// ---- POUs/20_AUTO/ST180/VISU_ST180.TcVIS
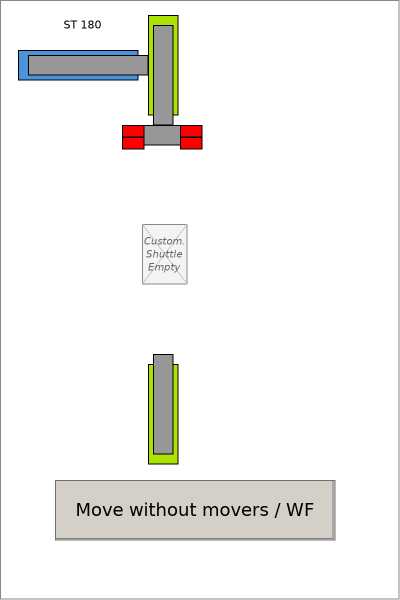
VISUALIZATION VISU_ST180  // 400x600
    Image (142,224 45x60), invisible if: NOT __ISVALIDREF(GVL.st180_aut._Mover), image: Custom.Shuttle Empty
    Rectangle (18,50 120x30)
    Rectangle (28,55 120x20)
        p3560616238: GVL.st180_aut.fb_Pnp.fb_simu_axis180_01Y.rOUT_PixActual
    Rectangle (148,15 30x100)
        p3560616238: GVL.st180_aut.fb_Pnp.fb_simu_axis180_01Y.rOUT_PixActual
    Rectangle (153,25 20x100)
        p2738717112: GVL.st180_aut.fb_Pnp.fb_simu_axis180_02Z.rOUT_PixActual
        p3560616238: GVL.st180_aut.fb_Pnp.fb_simu_axis180_01Y.rOUT_PixActual
    Label (40,15 85x20), "ST 180"
    Rectangle (122,125 80x20)
        p2738717112: GVL.st180_aut.fb_Pnp.fb_simu_axis180_02Z.rOUT_PixActual
        p3560616238: GVL.st180_aut.fb_Pnp.fb_simu_axis180_01Y.rOUT_PixActual
    Ellipse (123,125 20x20), colour toggle: GVL.st180_aut.fb_Pnp.fb_griperLeft.xIN_GS
        p3560616238: GVL.st180_aut.fb_Pnp.fb_simu_axis180_01Y.rOUT_PixActual
        p2738717112: GVL.st180_aut.fb_Pnp.fb_simu_axis180_02Z.rOUT_PixActual
    Ellipse (181,125 20x20), colour toggle: GVL.st180_aut.fb_Pnp.fb_griperRight.xIN_GS
        p3560616238: GVL.st180_aut.fb_Pnp.fb_simu_axis180_01Y.rOUT_PixActual
        p2738717112: GVL.st180_aut.fb_Pnp.fb_simu_axis180_02Z.rOUT_PixActual
    Rectangle (122,125 22x12), invisible if: NOT GVL.st180_aut.fb_Pnp.fb_clampLeft.xIN_GS
        p3560616238: GVL.st180_aut.fb_Pnp.fb_simu_axis180_01Y.rOUT_PixActual
        p2738717112: GVL.st180_aut.fb_Pnp.fb_simu_axis180_02Z.rOUT_PixActual
    Rectangle (180,125 22x12), invisible if: NOT GVL.st180_aut.fb_Pnp.fb_clampRight.xIN_GS
        p3560616238: GVL.st180_aut.fb_Pnp.fb_simu_axis180_01Y.rOUT_PixActual
        p2738717112: GVL.st180_aut.fb_Pnp.fb_simu_axis180_02Z.rOUT_PixActual
    Rectangle (122,137 22x12), invisible if: NOT GVL.st180_aut.fb_Pnp.fb_clampLeft.xIN_AS
        p3560616238: GVL.st180_aut.fb_Pnp.fb_simu_axis180_01Y.rOUT_PixActual
        p2738717112: GVL.st180_aut.fb_Pnp.fb_simu_axis180_02Z.rOUT_PixActual
    Rectangle (180,137 22x12), invisible if: NOT GVL.st180_aut.fb_Pnp.fb_clampRight.xIN_AS
        p3560616238: GVL.st180_aut.fb_Pnp.fb_simu_axis180_01Y.rOUT_PixActual
        p2738717112: GVL.st180_aut.fb_Pnp.fb_simu_axis180_02Z.rOUT_PixActual
    Rectangle (148,364 30x100)
    Rectangle (153,354 20x100)
        p2738717112: -GVL.st180_aut.fb_Pnp.fb_simu_axis180_10Z.rOUT_PixActual
    Button (55,480 280x60), "Move without movers / WF", colour toggle: HMI.bArForceCyclusState[StationList_e.ST180]
        tap HMI.btArForceCyclus[StationList_e.ST180].button
END_VISUALIZATION

// ---- POUs/20_AUTO/ST185/VISU_ST185.TcVIS
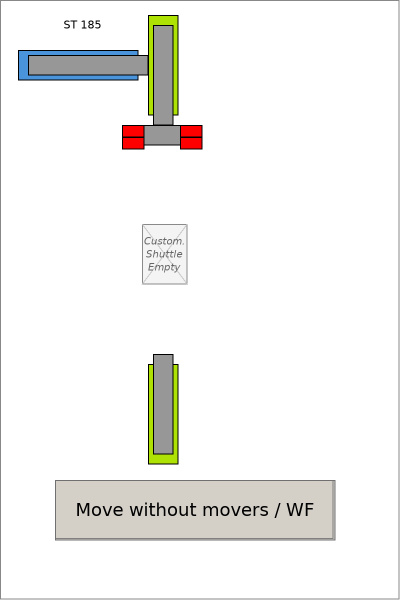
VISUALIZATION VISU_ST185  // 400x600
    Image (142,224 45x60), invisible if: NOT __ISVALIDREF(GVL.st185_aut._Mover), image: Custom.Shuttle Empty
    Rectangle (18,50 120x30)
    Rectangle (28,55 120x20)
        p3560616238: GVL.st185_aut.fb_Pnp.fb_simu_axis185_01Y.rOUT_PixActual
    Rectangle (148,15 30x100)
        p3560616238: GVL.st185_aut.fb_Pnp.fb_simu_axis185_01Y.rOUT_PixActual
    Rectangle (153,25 20x100)
        p2738717112: GVL.st185_aut.fb_Pnp.fb_simu_axis185_02Z.rOUT_PixActual
        p3560616238: GVL.st185_aut.fb_Pnp.fb_simu_axis185_01Y.rOUT_PixActual
    Label (40,15 85x20), "ST 185"
    Rectangle (122,125 80x20)
        p2738717112: GVL.st185_aut.fb_Pnp.fb_simu_axis185_02Z.rOUT_PixActual
        p3560616238: GVL.st185_aut.fb_Pnp.fb_simu_axis185_01Y.rOUT_PixActual
    Ellipse (123,125 20x20), colour toggle: GVL.st185_aut.fb_Pnp.fb_griperLeft.xIN_GS
        p3560616238: GVL.st185_aut.fb_Pnp.fb_simu_axis185_01Y.rOUT_PixActual
        p2738717112: GVL.st185_aut.fb_Pnp.fb_simu_axis185_02Z.rOUT_PixActual
    Ellipse (181,125 20x20), colour toggle: GVL.st185_aut.fb_Pnp.fb_griperRight.xIN_GS
        p3560616238: GVL.st185_aut.fb_Pnp.fb_simu_axis185_01Y.rOUT_PixActual
        p2738717112: GVL.st185_aut.fb_Pnp.fb_simu_axis185_02Z.rOUT_PixActual
    Rectangle (122,125 22x12), invisible if: NOT GVL.st185_aut.fb_Pnp.fb_clampLeft.xIN_GS
        p3560616238: GVL.st185_aut.fb_Pnp.fb_simu_axis185_01Y.rOUT_PixActual
        p2738717112: GVL.st185_aut.fb_Pnp.fb_simu_axis185_02Z.rOUT_PixActual
    Rectangle (180,125 22x12), invisible if: NOT GVL.st185_aut.fb_Pnp.fb_clampRight.xIN_GS
        p3560616238: GVL.st185_aut.fb_Pnp.fb_simu_axis185_01Y.rOUT_PixActual
        p2738717112: GVL.st185_aut.fb_Pnp.fb_simu_axis185_02Z.rOUT_PixActual
    Rectangle (122,137 22x12), invisible if: NOT GVL.st185_aut.fb_Pnp.fb_clampLeft.xIN_AS
        p3560616238: GVL.st185_aut.fb_Pnp.fb_simu_axis185_01Y.rOUT_PixActual
        p2738717112: GVL.st185_aut.fb_Pnp.fb_simu_axis185_02Z.rOUT_PixActual
    Rectangle (180,137 22x12), invisible if: NOT GVL.st185_aut.fb_Pnp.fb_clampRight.xIN_AS
        p3560616238: GVL.st185_aut.fb_Pnp.fb_simu_axis185_01Y.rOUT_PixActual
        p2738717112: GVL.st185_aut.fb_Pnp.fb_simu_axis185_02Z.rOUT_PixActual
    Rectangle (148,364 30x100)
    Rectangle (153,354 20x100)
        p2738717112: -GVL.st185_aut.fb_Pnp.fb_simu_axis185_10Z.rOUT_PixActual
    Button (55,480 280x60), "Move without movers / WF", colour toggle: HMI.bArForceCyclusState[StationList_e.ST185]
        tap HMI.btArForceCyclus[StationList_e.ST185].button
END_VISUALIZATION
